Universal Robots PolyScope program: L04_force.urp

Program L04_force (installation=default directory=/programs createdIn=5.9.1.1031110 lastSavedIn=5.9.1.1031110 robotSerialNumber=20195501059)
Calibrated DH parameters: a=[0.000146, -0.418764, -0.053981, 0.000058, -0.000023, 0]; d=[0.162545, 37.319448, -206.067439, 168.881546, 0.09955, 0.099464]; alpha=[1.57004, -0.001979, 0.002304, 1.570607, -1.57066, 0]; deltaTheta=[0, -0.174616, -1.258233, 1.432844, -0.000001, 0]
BeforeStart
  start_p := get_actual_tcp_pose()
  MoveL speed 250 mm/s, acceleration 1200 mm/s^2 (useActiveTCP=true) feature=Base
    Waypoint Waypoint (Variable): variable=start_p
Robot Program (runOnlyOnce=true)
  MoveL speed 250 mm/s, acceleration 1200 mm/s^2 (useActiveTCP=true) feature=Base
    Waypoint approach_p: TCP in base x=361.881 y=-355.664 z=37.792 mm, rx=2.2092 ry=2.2334 rz=-0.0001 rad; joints [120.211, -76.405, 118.753, -132.349, 270.051, 119.629] deg; TCP offset x=0 y=0 z=174 mm, rx=0 ry=0 rz=0 rad
    MoveDirectionNode (selectedDirection=ZMinus toolParams=0.01, 0.6)
      Until TOOL_CONTACT_DETECTION (allowActions=false retraction=0.006 decelerationAcceleration=2 decelerationAngularAcceleration=34.906585)
    URCap Force Control (Robotiq_Copilot, Robotiq Inc.) dataModel(NodeInitializedKey=true, force_x=0, force_y=0, force_mx=0, force_my=0, limit_x_neg=-100, limit_y_neg=-100, limit_z_neg=-100, limit_x_pos=100, limit_y_pos=100, limit_z_pos=100, limit_mx_neg=-20, limit_my_neg=-20, limit_mx_pos=20, limit_my_pos=20, stiffness_x=100, stiffness_y=100, stiffness_z_position=100, stiffness_mx=100, stiffness_my=100, stiffness_mz=100, adaptive_stiffness=true, is_force_control_about_actual_position=true, ft_control_z=true, ft_control_mz=true, limit_mz_neg=-90, limit_mz_pos=90, force_mz=0.5, ft_control_y=false, ft_control_mx=false, ft_control_my=false, HackTriggeringContributionIsDefinedMethodKey=true, ft_control_x=false, TranslatableFeatureKey=1, force_z=20)
      Wait Sleep waitTime=5
    Waypoint approach_p: TCP in base x=361.881 y=-355.664 z=37.792 mm, rx=2.2092 ry=2.2334 rz=-0.0001 rad; joints [120.211, -76.405, 118.753, -132.349, 270.051, 119.629] deg
